RESOURCE_TYPE ImageResource (* Resource Type *)
  (* Standard: 61499-2 *)
  (* Version 1.0, 2006-01-11, Anirudha, UoA, Moved to swing package *)
  (* Compiler header: package fb.rt.vhmi; import fb.rt.events.*; *)
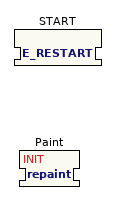
  FBS
    START : E_RESTART;
    Paint : repaint;
  END_FBS
END_RESOURCE_TYPE
